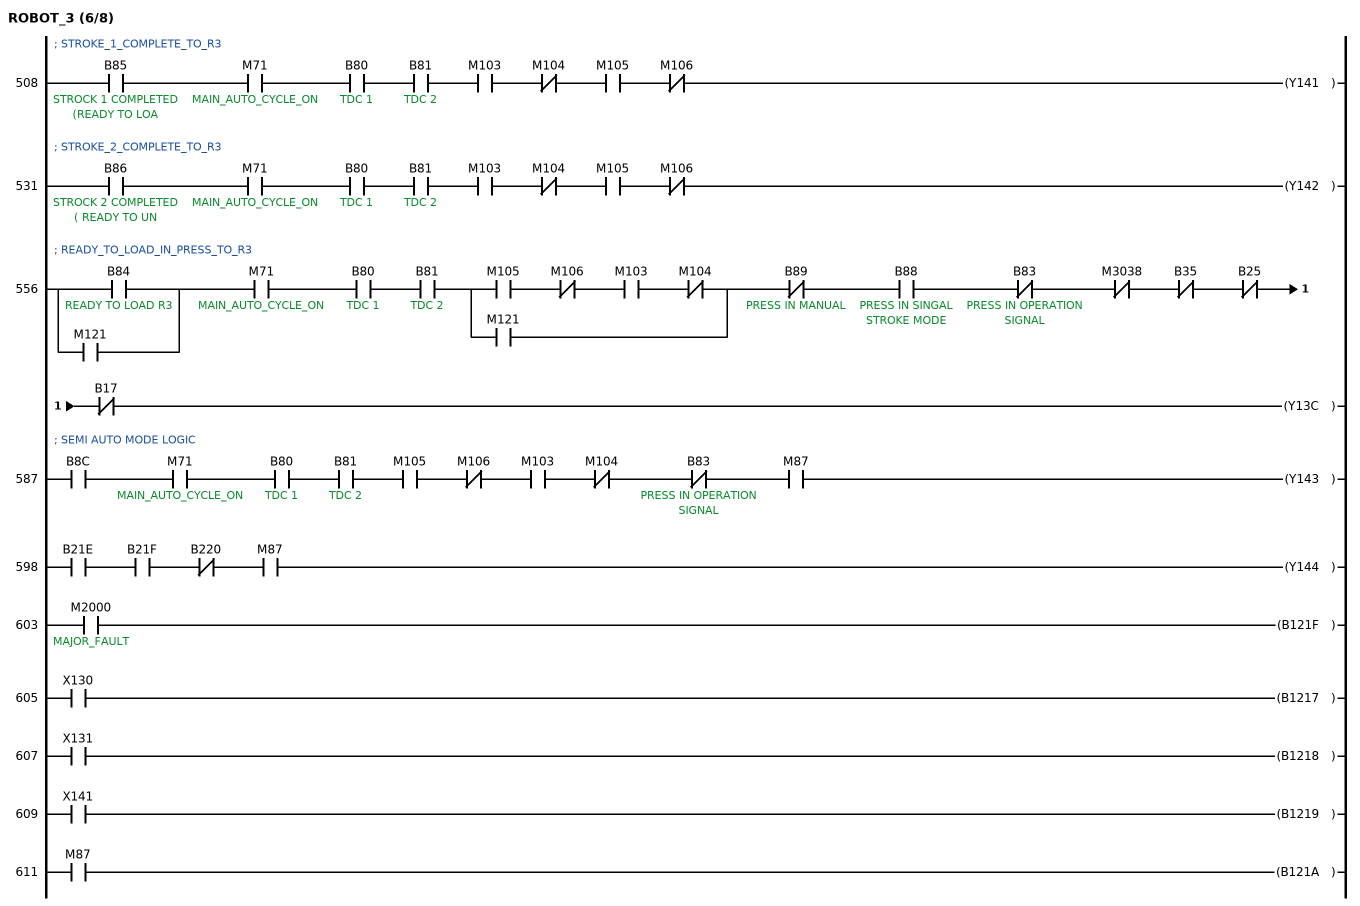
[picture p48: ladder of ROBOT_3, rungs at steps 508 to 611]
; STROKE_1_COMPLETE_TO_R3
508   LD      B85  ; STROCK 1 COMPLETED (READY TO LOA
      AND     M71  ; MAIN_AUTO_CYCLE_ON
      AND     B80  ; TDC 1
      AND     B81  ; TDC 2
      AND     M103
      ANI     M104
      AND     M105
      ANI     M106
      OUT     Y141
; STROKE_2_COMPLETE_TO_R3
531   LD      B86  ; STROCK 2 COMPLETED ( READY TO UN
      AND     M71  ; MAIN_AUTO_CYCLE_ON
      AND     B80  ; TDC 1
      AND     B81  ; TDC 2
      AND     M103
      ANI     M104
      AND     M105
      ANI     M106
      OUT     Y142
; READY_TO_LOAD_IN_PRESS_TO_R3
556   LD      B84  ; READY TO LOAD R3
      OR      M121
      AND     M71  ; MAIN_AUTO_CYCLE_ON
      AND     B80  ; TDC 1
      AND     B81  ; TDC 2
      LD      M105
      ANI     M106
      AND     M103
      ANI     M104
      OR      M121
      ANB
      ANI     B89  ; PRESS IN MANUAL
      AND     B88  ; PRESS IN SINGAL STROKE MODE
      ANI     B83  ; PRESS IN OPERATION SIGNAL
      ANI     M3038
      ANI     B35
      ANI     B25
      ANI     B17
      OUT     Y13C
; SEMI AUTO MODE LOGIC
587   LD      B8C
      AND     M71  ; MAIN_AUTO_CYCLE_ON
      AND     B80  ; TDC 1
      AND     B81  ; TDC 2
      AND     M105
      ANI     M106
      AND     M103
      ANI     M104
      ANI     B83  ; PRESS IN OPERATION SIGNAL
      AND     M87
      OUT     Y143
598   LD      B21E
      AND     B21F
      ANI     B220
      AND     M87
      OUT     Y144
603   LD      M2000  ; MAJOR_FAULT
      OUT     B121F
605   LD      X130
      OUT     B1217
607   LD      X131
      OUT     B1218
609   LD      X141
      OUT     B1219
611   LD      M87
      OUT     B121A
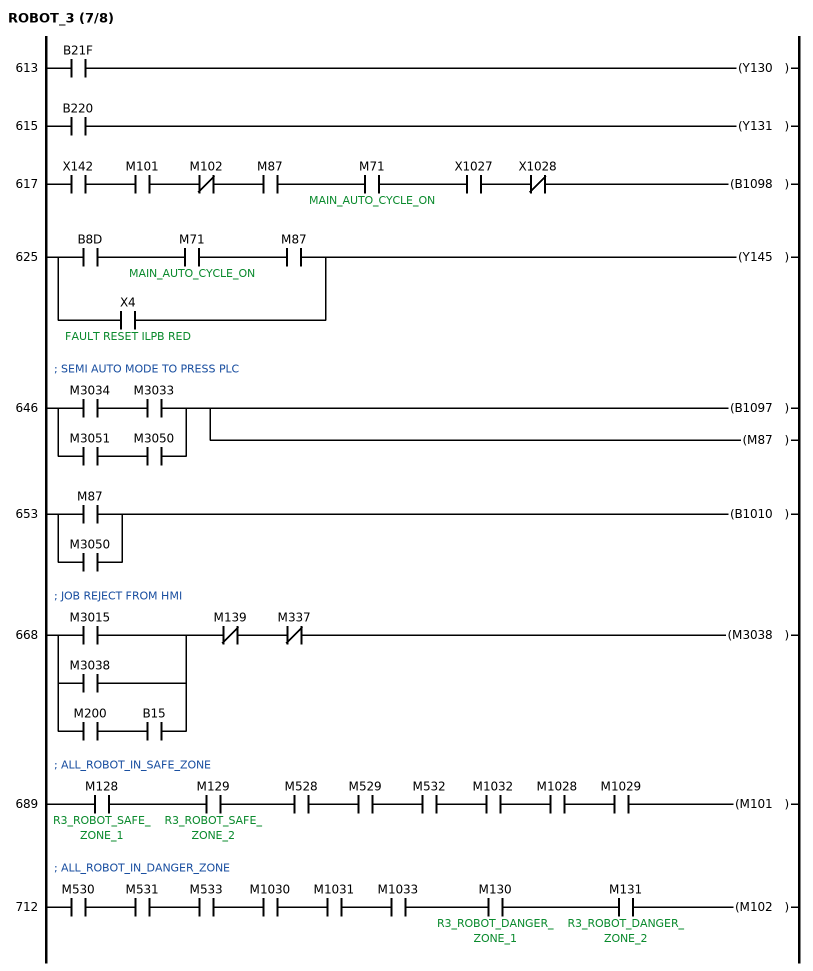
613   LD      B21F
      OUT     Y130
615   LD      B220
      OUT     Y131
617   LD      X142
      AND     M101
      ANI     M102
      AND     M87
      AND     M71  ; MAIN_AUTO_CYCLE_ON
      AND     X1027
      ANI     X1028
      OUT     B1098
625   LD      B8D
      AND     M71  ; MAIN_AUTO_CYCLE_ON
      AND     M87
      OR      X4  ; FAULT RESET ILPB RED
      OUT     Y145
; SEMI AUTO MODE TO PRESS PLC
646   LD      M3034
      AND     M3033
      LD      M3051
      AND     M3050
      ORB
      OUT     B1097
      OUT     M87
653   LD      M87
      OR      M3050
      OUT     B1010
; JOB REJECT FROM HMI
668   LD      M3015
      OR      M3038
      LD      M200
      AND     B15
      ORB
      ANI     M139
      ANI     M337
      OUT     M3038
; ALL_ROBOT_IN_SAFE_ZONE
689   LD      M128  ; R3_ROBOT_SAFE_ZONE_1
      AND     M129  ; R3_ROBOT_SAFE_ZONE_2
      AND     M528
      AND     M529
      AND     M532
      AND     M1032
      AND     M1028
      AND     M1029
      OUT     M101
; ALL_ROBOT_IN_DANGER_ZONE
712   LD      M530
      AND     M531
      AND     M533
      AND     M1030
      AND     M1031
      AND     M1033
      AND     M130  ; R3_ROBOT_DANGER_ZONE_1
      AND     M131  ; R3_ROBOT_DANGER_ZONE_2
      OUT     M102
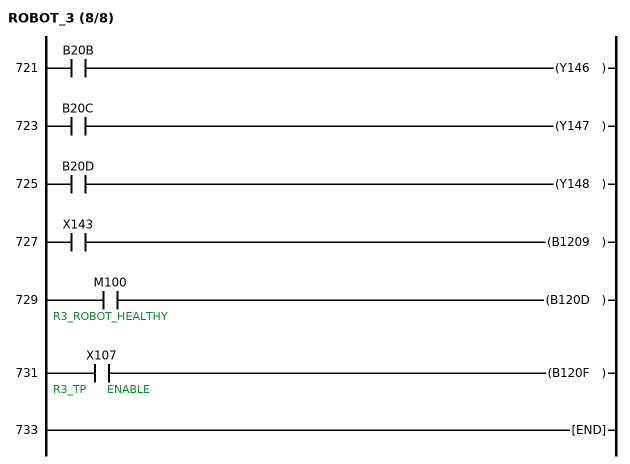
721   LD      B20B
      OUT     Y146
723   LD      B20C
      OUT     Y147
725   LD      B20D
      OUT     Y148
727   LD      X143
      OUT     B1209
729   LD      M100  ; R3_ROBOT_HEALTHY
      OUT     B120D
731   LD      X107  ; R3_TP      ENABLE
      OUT     B120F
733   END
END_PROGRAM

PROGRAM ROBOT_4
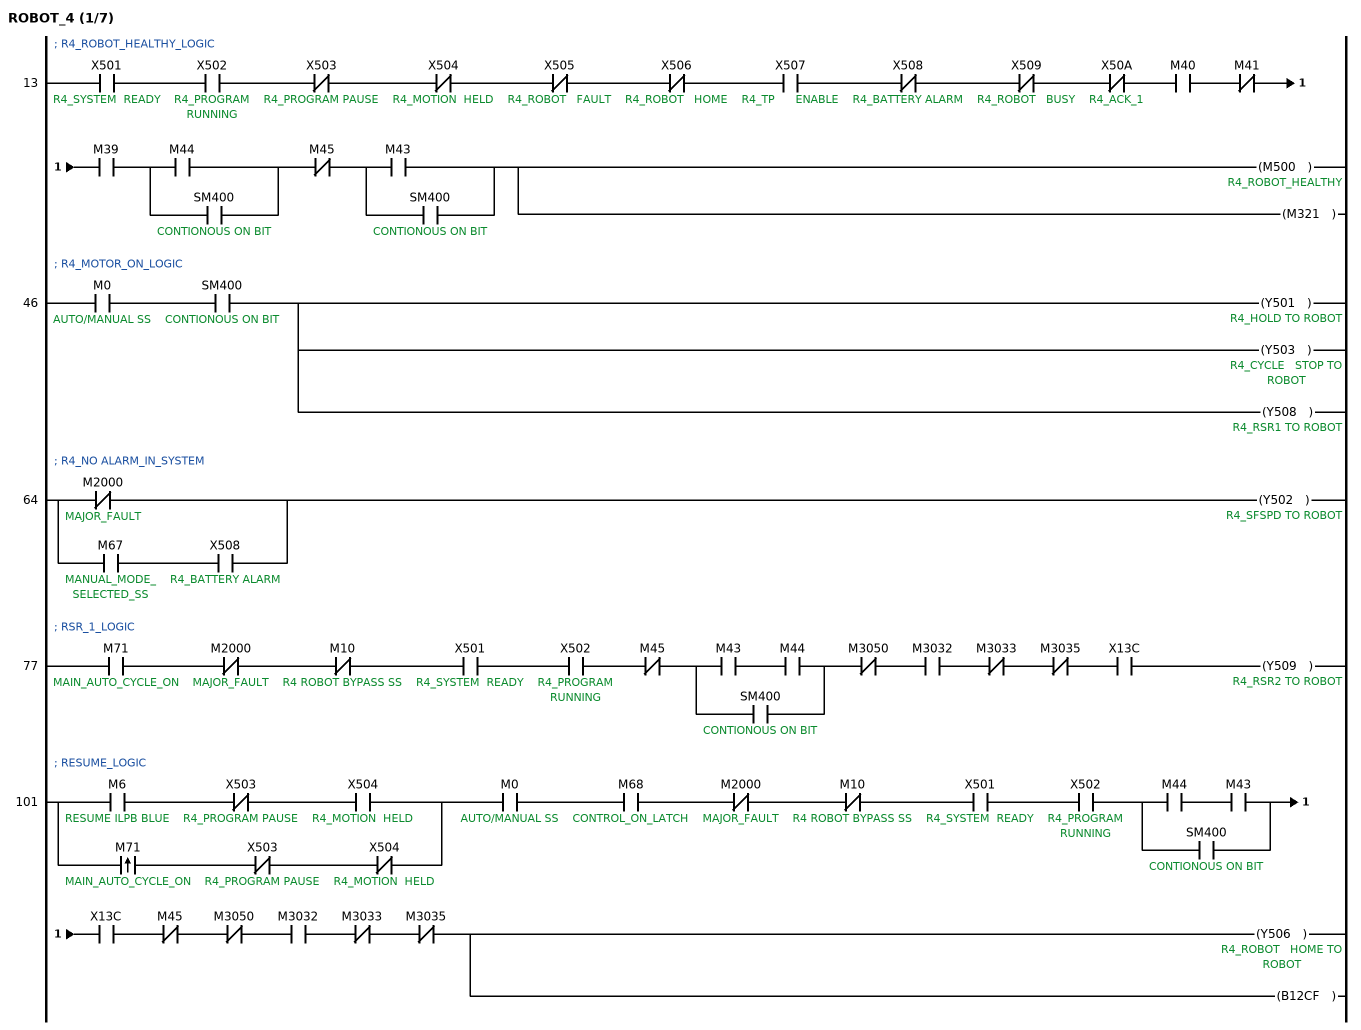
; R4_ROBOT_HEALTHY_LOGIC
13    LD      X501  ; R4_SYSTEM  READY
      AND     X502  ; R4_PROGRAM RUNNING
      ANI     X503  ; R4_PROGRAM PAUSE
      ANI     X504  ; R4_MOTION  HELD
      ANI     X505  ; R4_ROBOT   FAULT
      ANI     X506  ; R4_ROBOT   HOME
      AND     X507  ; R4_TP      ENABLE
      ANI     X508  ; R4_BATTERY ALARM
      ANI     X509  ; R4_ROBOT   BUSY
      ANI     X50A  ; R4_ACK_1
      AND     M40
      ANI     M41
      AND     M39
      LD      M44
      OR      SM400  ; CONTIONOUS ON BIT
      ANB
      ANI     M45
      LD      M43
      OR      SM400  ; CONTIONOUS ON BIT
      ANB
      OUT     M500  ; R4_ROBOT_HEALTHY
      OUT     M321
; R4_MOTOR_ON_LOGIC
46    LD      M0  ; AUTO/MANUAL SS
      AND     SM400  ; CONTIONOUS ON BIT
      OUT     Y501  ; R4_HOLD TO ROBOT
      OUT     Y503  ; R4_CYCLE   STOP TO ROBOT
      OUT     Y508  ; R4_RSR1 TO ROBOT
; R4_NO ALARM_IN_SYSTEM
64    LDI     M2000  ; MAJOR_FAULT
      LD      M67  ; MANUAL_MODE_SELECTED_SS
      AND     X508  ; R4_BATTERY ALARM
      ORB
      OUT     Y502  ; R4_SFSPD TO ROBOT
; RSR_1_LOGIC
77    LD      M71  ; MAIN_AUTO_CYCLE_ON
      ANI     M2000  ; MAJOR_FAULT
      ANI     M10  ; R4 ROBOT BYPASS SS
      AND     X501  ; R4_SYSTEM  READY
      AND     X502  ; R4_PROGRAM RUNNING
      ANI     M45
      LD      M43
      AND     M44
      OR      SM400  ; CONTIONOUS ON BIT
      ANB
      ANI     M3050
      AND     M3032
      ANI     M3033
      ANI     M3035
      AND     X13C
      OUT     Y509  ; R4_RSR2 TO ROBOT
; RESUME_LOGIC
101   LD      M6  ; RESUME ILPB BLUE
      ANI     X503  ; R4_PROGRAM PAUSE
      AND     X504  ; R4_MOTION  HELD
      LDP     M71  ; MAIN_AUTO_CYCLE_ON
      ANI     X503  ; R4_PROGRAM PAUSE
      ANI     X504  ; R4_MOTION  HELD
      ORB
      AND     M0  ; AUTO/MANUAL SS
      AND     M68  ; CONTROL_ON_LATCH
      ANI     M2000  ; MAJOR_FAULT
      ANI     M10  ; R4 ROBOT BYPASS SS
      AND     X501  ; R4_SYSTEM  READY
      AND     X502  ; R4_PROGRAM RUNNING
      LD      M44
      AND     M43
      OR      SM400  ; CONTIONOUS ON BIT
      ANB
      AND     X13C
      ANI     M45
      ANI     M3050
      AND     M3032
      ANI     M3033
      ANI     M3035
      OUT     Y506  ; R4_ROBOT   HOME TO ROBOT
      OUT     B12CF
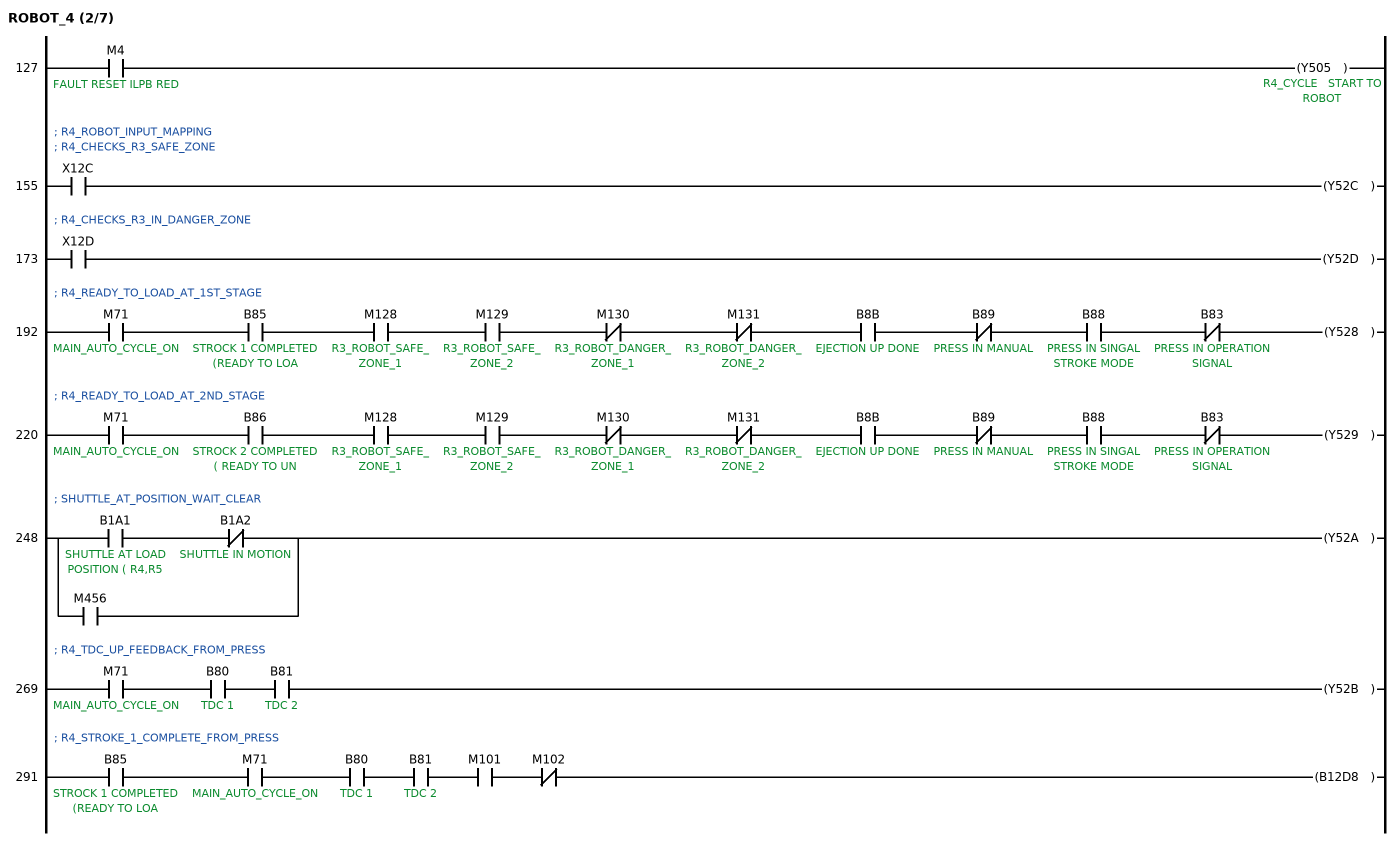
127   LD      M4  ; FAULT RESET ILPB RED
      OUT     Y505  ; R4_CYCLE   START TO ROBOT
; R4_ROBOT_INPUT_MAPPING
; R4_CHECKS_R3_SAFE_ZONE
155   LD      X12C
      OUT     Y52C
; R4_CHECKS_R3_IN_DANGER_ZONE
173   LD      X12D
      OUT     Y52D
; R4_READY_TO_LOAD_AT_1ST_STAGE
192   LD      M71  ; MAIN_AUTO_CYCLE_ON
      AND     B85  ; STROCK 1 COMPLETED (READY TO LOA
      AND     M128  ; R3_ROBOT_SAFE_ZONE_1
      AND     M129  ; R3_ROBOT_SAFE_ZONE_2
      ANI     M130  ; R3_ROBOT_DANGER_ZONE_1
      ANI     M131  ; R3_ROBOT_DANGER_ZONE_2
      AND     B8B  ; EJECTION UP DONE
      ANI     B89  ; PRESS IN MANUAL
      AND     B88  ; PRESS IN SINGAL STROKE MODE
      ANI     B83  ; PRESS IN OPERATION SIGNAL
      OUT     Y528
; R4_READY_TO_LOAD_AT_2ND_STAGE
220   LD      M71  ; MAIN_AUTO_CYCLE_ON
      AND     B86  ; STROCK 2 COMPLETED ( READY TO UN
      AND     M128  ; R3_ROBOT_SAFE_ZONE_1
      AND     M129  ; R3_ROBOT_SAFE_ZONE_2
      ANI     M130  ; R3_ROBOT_DANGER_ZONE_1
      ANI     M131  ; R3_ROBOT_DANGER_ZONE_2
      AND     B8B  ; EJECTION UP DONE
      ANI     B89  ; PRESS IN MANUAL
      AND     B88  ; PRESS IN SINGAL STROKE MODE
      ANI     B83  ; PRESS IN OPERATION SIGNAL
      OUT     Y529
; SHUTTLE_AT_POSITION_WAIT_CLEAR
248   LD      B1A1  ; SHUTTLE AT LOAD POSITION ( R4,R5
      ANI     B1A2  ; SHUTTLE IN MOTION
      OR      M456
      OUT     Y52A
; R4_TDC_UP_FEEDBACK_FROM_PRESS
269   LD      M71  ; MAIN_AUTO_CYCLE_ON
      AND     B80  ; TDC 1
      AND     B81  ; TDC 2
      OUT     Y52B
; R4_STROKE_1_COMPLETE_FROM_PRESS
291   LD      B85  ; STROCK 1 COMPLETED (READY TO LOA
      AND     M71  ; MAIN_AUTO_CYCLE_ON
      AND     B80  ; TDC 1
      AND     B81  ; TDC 2
      AND     M101
      ANI     M102
      OUT     B12D8
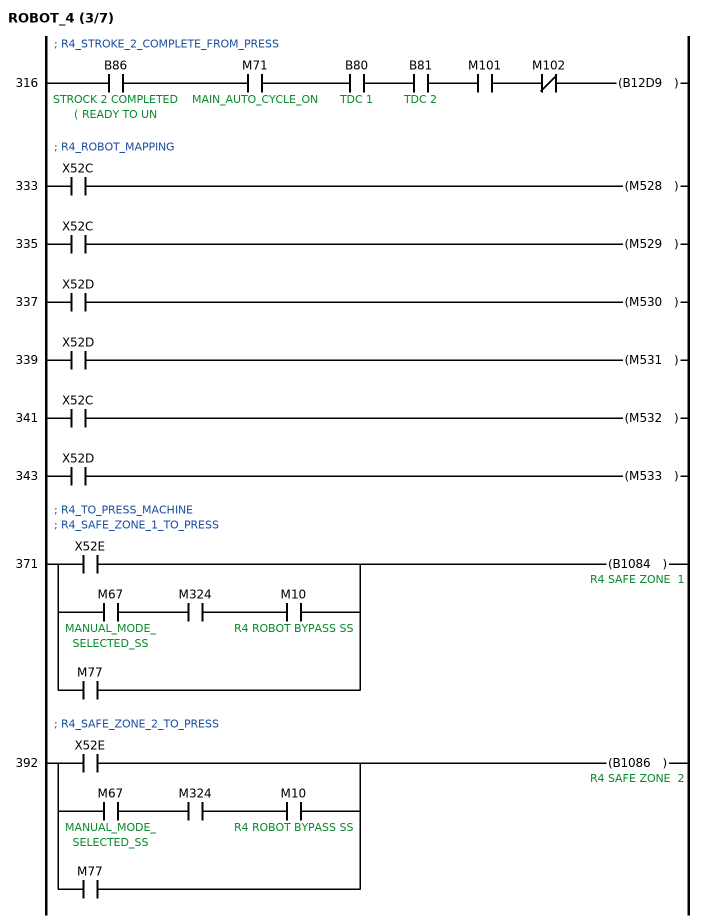
; R4_STROKE_2_COMPLETE_FROM_PRESS
316   LD      B86  ; STROCK 2 COMPLETED ( READY TO UN
      AND     M71  ; MAIN_AUTO_CYCLE_ON
      AND     B80  ; TDC 1
      AND     B81  ; TDC 2
      AND     M101
      ANI     M102
      OUT     B12D9
; R4_ROBOT_MAPPING
333   LD      X52C
      OUT     M528
335   LD      X52C
      OUT     M529
337   LD      X52D
      OUT     M530
339   LD      X52D
      OUT     M531
341   LD      X52C
      OUT     M532
343   LD      X52D
      OUT     M533
; R4_TO_PRESS_MACHINE
; R4_SAFE_ZONE_1_TO_PRESS
371   LD      X52E
      LD      M67  ; MANUAL_MODE_SELECTED_SS
      AND     M324
      AND     M10  ; R4 ROBOT BYPASS SS
      ORB
      OR      M77
      OUT     B1084  ; R4 SAFE ZONE  1
; R4_SAFE_ZONE_2_TO_PRESS
392   LD      X52E
      LD      M67  ; MANUAL_MODE_SELECTED_SS
      AND     M324
      AND     M10  ; R4 ROBOT BYPASS SS
      ORB
      OR      M77
      OUT     B1086  ; R4 SAFE ZONE  2
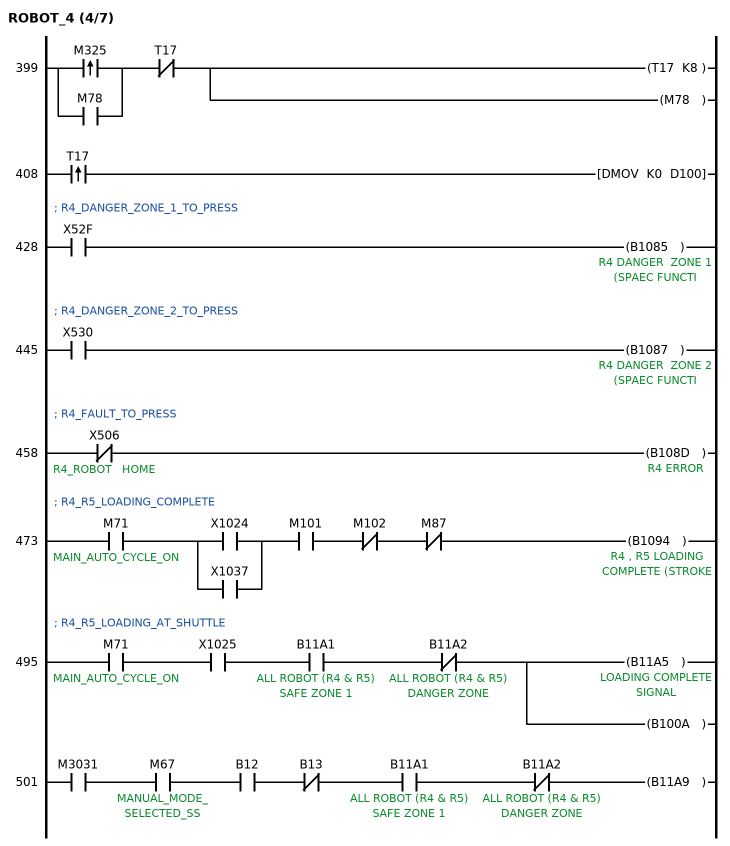
399   LDP     M325
      OR      M78
      ANI     T17
      OUT     T17 K8
      OUT     M78
408   LDP     T17
      DMOV    K0 D100
; R4_DANGER_ZONE_1_TO_PRESS
428   LD      X52F
      OUT     B1085  ; R4 DANGER  ZONE 1 (SPAEC FUNCTI
; R4_DANGER_ZONE_2_TO_PRESS
445   LD      X530
      OUT     B1087  ; R4 DANGER  ZONE 2 (SPAEC FUNCTI
; R4_FAULT_TO_PRESS
458   LDI     X506  ; R4_ROBOT   HOME
      OUT     B108D  ; R4 ERROR
; R4_R5_LOADING_COMPLETE
473   LD      M71  ; MAIN_AUTO_CYCLE_ON
      LD      X1024
      OR      X1037
      ANB
      AND     M101
      ANI     M102
      ANI     M87
      OUT     B1094  ; R4 , R5 LOADING COMPLETE (STROKE
; R4_R5_LOADING_AT_SHUTTLE
495   LD      M71  ; MAIN_AUTO_CYCLE_ON
      AND     X1025
      AND     B11A1  ; ALL ROBOT (R4 & R5) SAFE ZONE 1
      ANI     B11A2  ; ALL ROBOT (R4 & R5) DANGER ZONE
      OUT     B11A5  ; LOADING COMPLETE SIGNAL
      OUT     B100A
501   LD      M3031
      AND     M67  ; MANUAL_MODE_SELECTED_SS
      AND     B12
      ANI     B13
      AND     B11A1  ; ALL ROBOT (R4 & R5) SAFE ZONE 1
      ANI     B11A2  ; ALL ROBOT (R4 & R5) DANGER ZONE
      OUT     B11A9
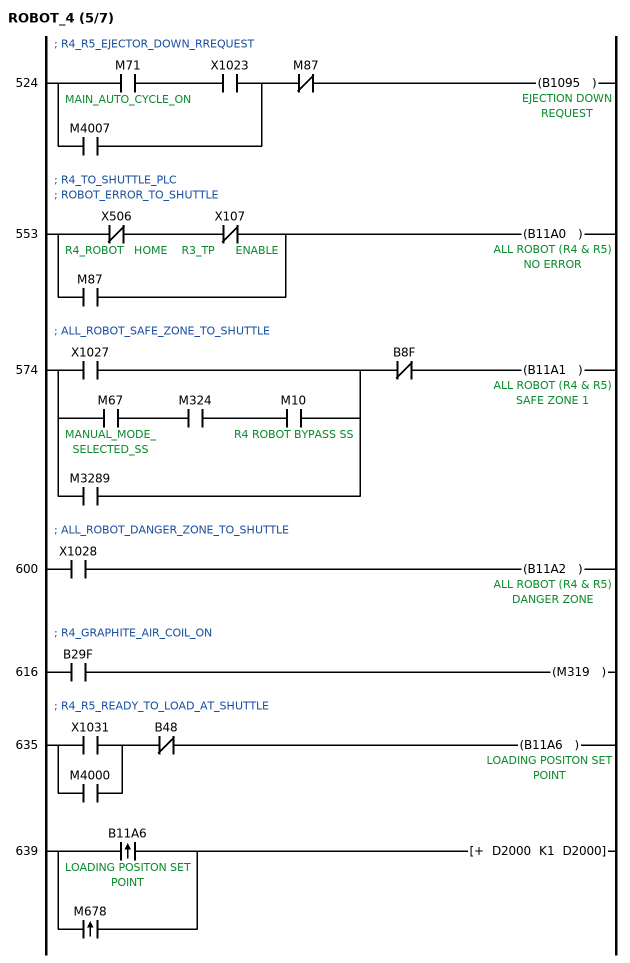
; R4_R5_EJECTOR_DOWN_RREQUEST
524   LD      M71  ; MAIN_AUTO_CYCLE_ON
      AND     X1023
      OR      M4007
      ANI     M87
      OUT     B1095  ; EJECTION DOWN REQUEST
; R4_TO_SHUTTLE_PLC
; ROBOT_ERROR_TO_SHUTTLE
553   LDI     X506  ; R4_ROBOT   HOME
      ANI     X107  ; R3_TP      ENABLE
      OR      M87
      OUT     B11A0  ; ALL ROBOT (R4 & R5) NO ERROR
; ALL_ROBOT_SAFE_ZONE_TO_SHUTTLE
574   LD      X1027
      LD      M67  ; MANUAL_MODE_SELECTED_SS
      AND     M324
      AND     M10  ; R4 ROBOT BYPASS SS
      ORB
      OR      M3289
      ANI     B8F
      OUT     B11A1  ; ALL ROBOT (R4 & R5) SAFE ZONE 1
; ALL_ROBOT_DANGER_ZONE_TO_SHUTTLE
600   LD      X1028
      OUT     B11A2  ; ALL ROBOT (R4 & R5) DANGER ZONE
; R4_GRAPHITE_AIR_COIL_ON
616   LD      B29F
      OUT     M319
; R4_R5_READY_TO_LOAD_AT_SHUTTLE
635   LD      X1031
      OR      M4000
      ANI     B48
      OUT     B11A6  ; LOADING POSITON SET POINT
639   LDP     B11A6  ; LOADING POSITON SET POINT
      ORP     M678
      +       D2000 K1 D2000
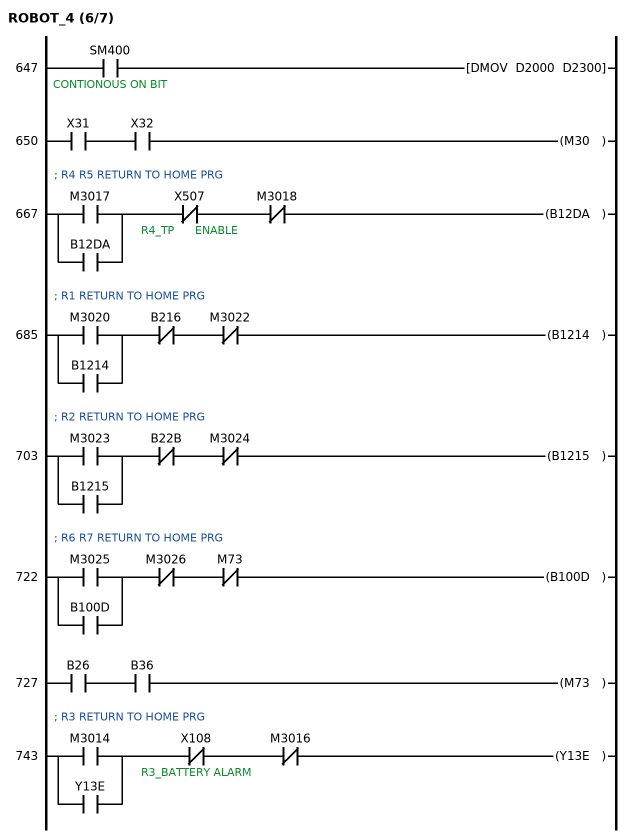
647   LD      SM400  ; CONTIONOUS ON BIT
      DMOV    D2000 D2300
650   LD      X31
      AND     X32
      OUT     M30
; R4 R5 RETURN TO HOME PRG
667   LD      M3017
      OR      B12DA
      ANI     X507  ; R4_TP      ENABLE
      ANI     M3018
      OUT     B12DA
; R1 RETURN TO HOME PRG
685   LD      M3020
      OR      B1214
      ANI     B216
      ANI     M3022
      OUT     B1214
; R2 RETURN TO HOME PRG
703   LD      M3023
      OR      B1215
      ANI     B22B
      ANI     M3024
      OUT     B1215
; R6 R7 RETURN TO HOME PRG
722   LD      M3025
      OR      B100D
      ANI     M3026
      ANI     M73
      OUT     B100D
727   LD      B26
      AND     B36
      OUT     M73
; R3 RETURN TO HOME PRG
743   LD      M3014
      OR      Y13E
      ANI     X108  ; R3_BATTERY ALARM
      ANI     M3016
      OUT     Y13E
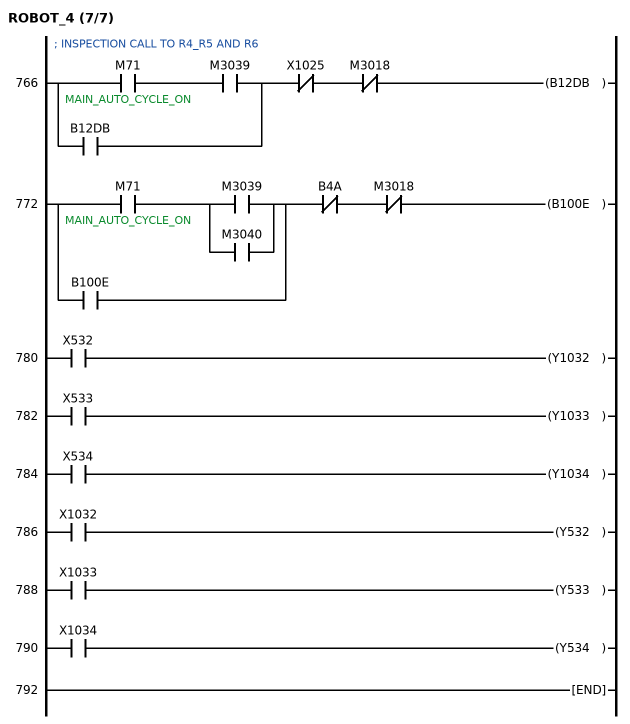
; INSPECTION CALL TO R4_R5 AND R6
766   LD      M71  ; MAIN_AUTO_CYCLE_ON
      AND     M3039
      OR      B12DB
      ANI     X1025
      ANI     M3018
      OUT     B12DB
772   LD      M71  ; MAIN_AUTO_CYCLE_ON
      LD      M3039
      OR      M3040
      ANB
      OR      B100E
      ANI     B4A
      ANI     M3018
      OUT     B100E
780   LD      X532
      OUT     Y1032
782   LD      X533
      OUT     Y1033
784   LD      X534
      OUT     Y1034
786   LD      X1032
      OUT     Y532
788   LD      X1033
      OUT     Y533
790   LD      X1034
      OUT     Y534
792   END
END_PROGRAM

PROGRAM ROBOT_5
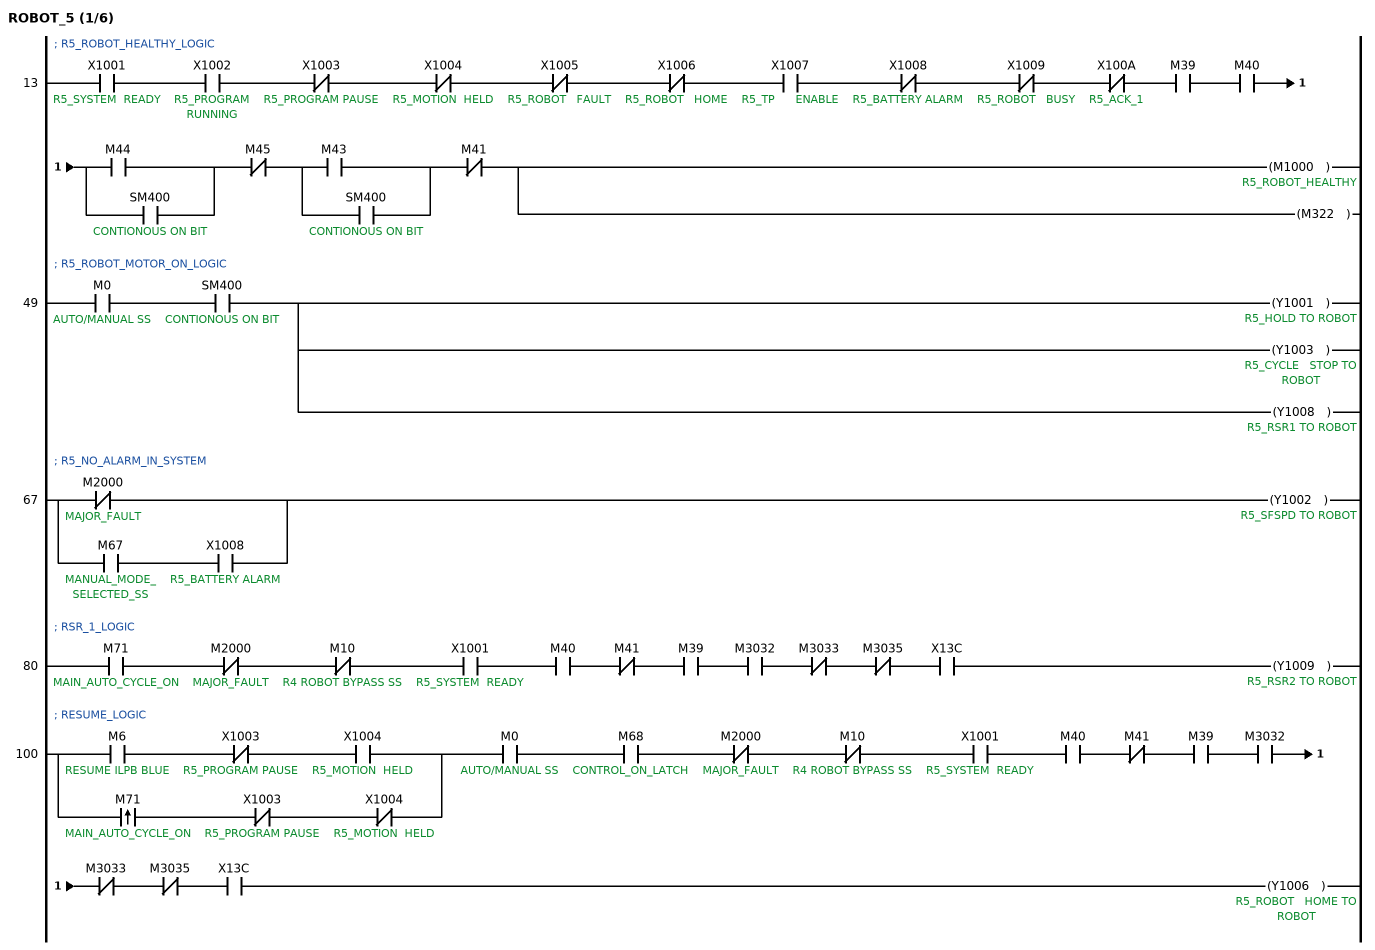
; R5_ROBOT_HEALTHY_LOGIC
13    LD      X1001  ; R5_SYSTEM  READY
      AND     X1002  ; R5_PROGRAM RUNNING
      ANI     X1003  ; R5_PROGRAM PAUSE
      ANI     X1004  ; R5_MOTION  HELD
      ANI     X1005  ; R5_ROBOT   FAULT
      ANI     X1006  ; R5_ROBOT   HOME
      AND     X1007  ; R5_TP      ENABLE
      ANI     X1008  ; R5_BATTERY ALARM
      ANI     X1009  ; R5_ROBOT   BUSY
      ANI     X100A  ; R5_ACK_1
      AND     M39
      AND     M40
      LD      M44
      OR      SM400  ; CONTIONOUS ON BIT
      ANB
      ANI     M45
      LD      M43
      OR      SM400  ; CONTIONOUS ON BIT
      ANB
      ANI     M41
      OUT     M1000  ; R5_ROBOT_HEALTHY
      OUT     M322
; R5_ROBOT_MOTOR_ON_LOGIC
49    LD      M0  ; AUTO/MANUAL SS
      AND     SM400  ; CONTIONOUS ON BIT
      OUT     Y1001  ; R5_HOLD TO ROBOT
      OUT     Y1003  ; R5_CYCLE   STOP TO ROBOT
      OUT     Y1008  ; R5_RSR1 TO ROBOT
; R5_NO_ALARM_IN_SYSTEM
67    LDI     M2000  ; MAJOR_FAULT
      LD      M67  ; MANUAL_MODE_SELECTED_SS
      AND     X1008  ; R5_BATTERY ALARM
      ORB
      OUT     Y1002  ; R5_SFSPD TO ROBOT
; RSR_1_LOGIC
80    LD      M71  ; MAIN_AUTO_CYCLE_ON
      ANI     M2000  ; MAJOR_FAULT
      ANI     M10  ; R4 ROBOT BYPASS SS
      AND     X1001  ; R5_SYSTEM  READY
      AND     M40
      ANI     M41
      AND     M39
      AND     M3032
      ANI     M3033
      ANI     M3035
      AND     X13C
      OUT     Y1009  ; R5_RSR2 TO ROBOT
; RESUME_LOGIC
100   LD      M6  ; RESUME ILPB BLUE
      ANI     X1003  ; R5_PROGRAM PAUSE
      AND     X1004  ; R5_MOTION  HELD
      LDP     M71  ; MAIN_AUTO_CYCLE_ON
      ANI     X1003  ; R5_PROGRAM PAUSE
      ANI     X1004  ; R5_MOTION  HELD
      ORB
      AND     M0  ; AUTO/MANUAL SS
      AND     M68  ; CONTROL_ON_LATCH
      ANI     M2000  ; MAJOR_FAULT
      ANI     M10  ; R4 ROBOT BYPASS SS
      AND     X1001  ; R5_SYSTEM  READY
      AND     M40
      ANI     M41
      AND     M39
      AND     M3032
      ANI     M3033
      ANI     M3035
      AND     X13C
      OUT     Y1006  ; R5_ROBOT   HOME TO ROBOT
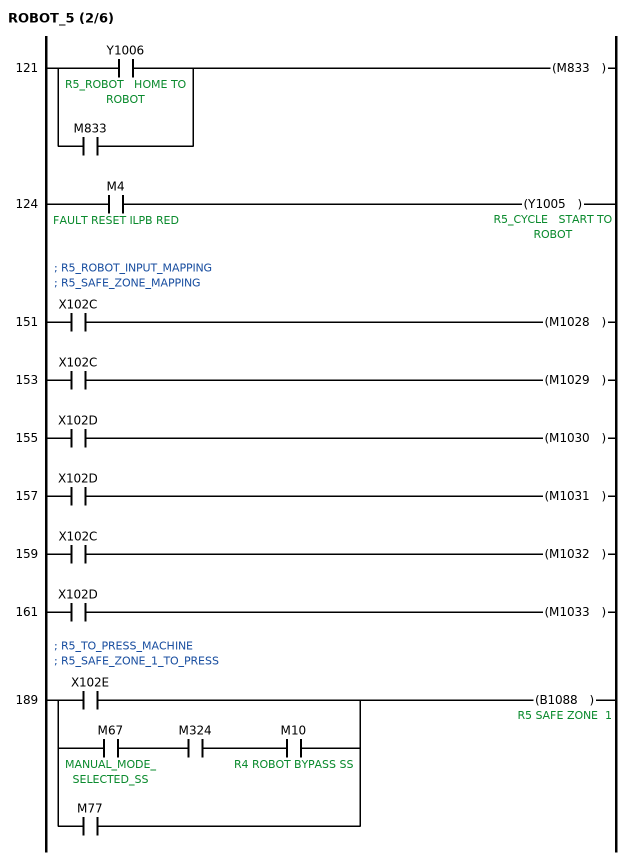
121   LD      Y1006  ; R5_ROBOT   HOME TO ROBOT
      OR      M833
      OUT     M833
124   LD      M4  ; FAULT RESET ILPB RED
      OUT     Y1005  ; R5_CYCLE   START TO ROBOT
; R5_ROBOT_INPUT_MAPPING
; R5_SAFE_ZONE_MAPPING
151   LD      X102C
      OUT     M1028
153   LD      X102C
      OUT     M1029
155   LD      X102D
      OUT     M1030
157   LD      X102D
      OUT     M1031
159   LD      X102C
      OUT     M1032
161   LD      X102D
      OUT     M1033
; R5_TO_PRESS_MACHINE
; R5_SAFE_ZONE_1_TO_PRESS
189   LD      X102E
      LD      M67  ; MANUAL_MODE_SELECTED_SS
      AND     M324
      AND     M10  ; R4 ROBOT BYPASS SS
      ORB
      OR      M77
      OUT     B1088  ; R5 SAFE ZONE  1
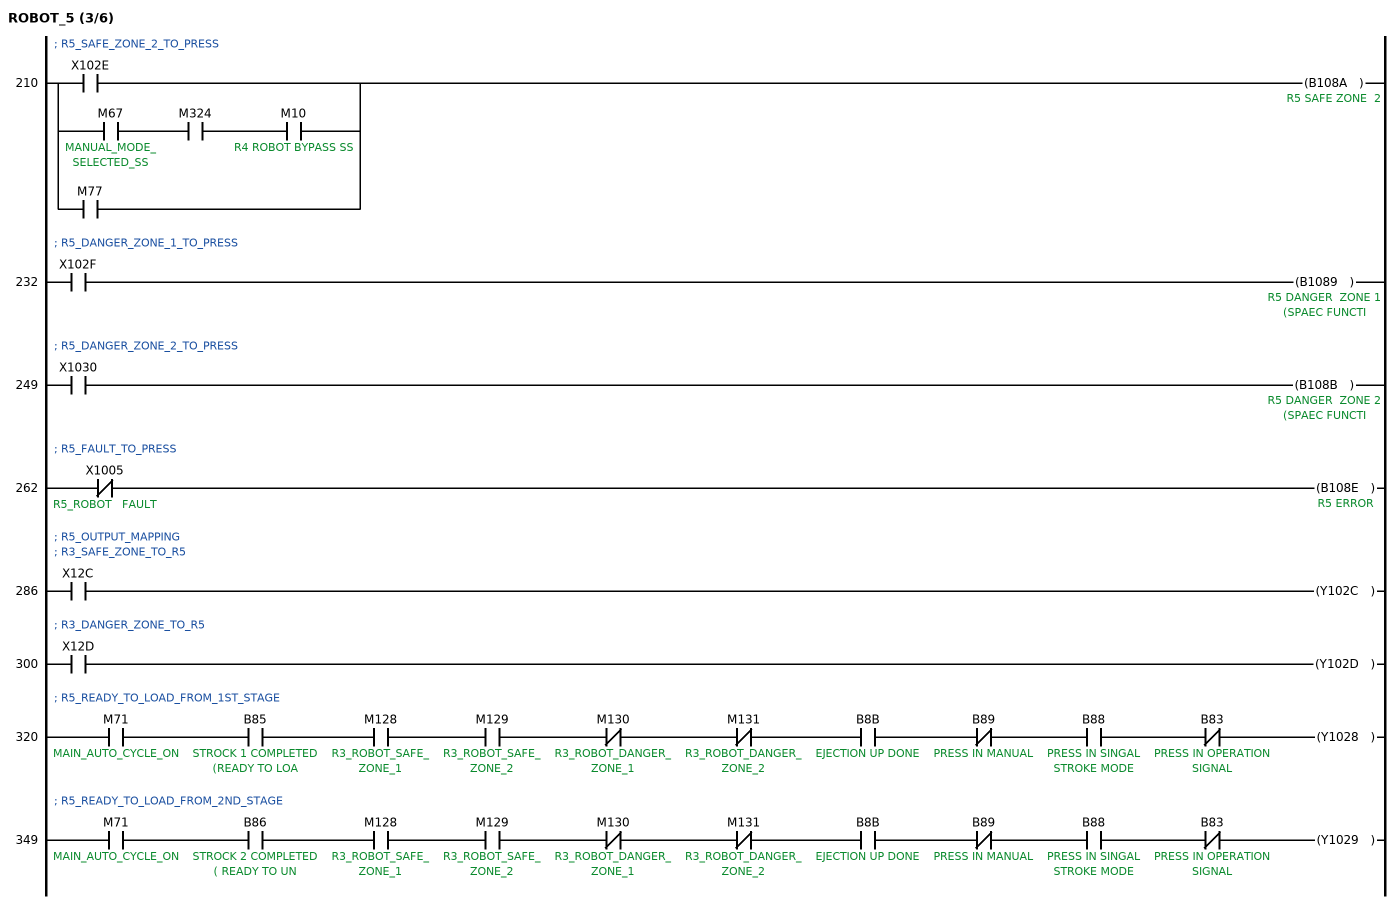
; R5_SAFE_ZONE_2_TO_PRESS
210   LD      X102E
      LD      M67  ; MANUAL_MODE_SELECTED_SS
      AND     M324
      AND     M10  ; R4 ROBOT BYPASS SS
      ORB
      OR      M77
      OUT     B108A  ; R5 SAFE ZONE  2
; R5_DANGER_ZONE_1_TO_PRESS
232   LD      X102F
      OUT     B1089  ; R5 DANGER  ZONE 1 (SPAEC FUNCTI
; R5_DANGER_ZONE_2_TO_PRESS
249   LD      X1030
      OUT     B108B  ; R5 DANGER  ZONE 2 (SPAEC FUNCTI
; R5_FAULT_TO_PRESS
262   LDI     X1005  ; R5_ROBOT   FAULT
      OUT     B108E  ; R5 ERROR
; R5_OUTPUT_MAPPING
; R3_SAFE_ZONE_TO_R5
286   LD      X12C
      OUT     Y102C
; R3_DANGER_ZONE_TO_R5
300   LD      X12D
      OUT     Y102D
; R5_READY_TO_LOAD_FROM_1ST_STAGE
320   LD      M71  ; MAIN_AUTO_CYCLE_ON
      AND     B85  ; STROCK 1 COMPLETED (READY TO LOA
      AND     M128  ; R3_ROBOT_SAFE_ZONE_1
      AND     M129  ; R3_ROBOT_SAFE_ZONE_2
      ANI     M130  ; R3_ROBOT_DANGER_ZONE_1
      ANI     M131  ; R3_ROBOT_DANGER_ZONE_2
      AND     B8B  ; EJECTION UP DONE
      ANI     B89  ; PRESS IN MANUAL
      AND     B88  ; PRESS IN SINGAL STROKE MODE
      ANI     B83  ; PRESS IN OPERATION SIGNAL
      OUT     Y1028
; R5_READY_TO_LOAD_FROM_2ND_STAGE
349   LD      M71  ; MAIN_AUTO_CYCLE_ON
      AND     B86  ; STROCK 2 COMPLETED ( READY TO UN
      AND     M128  ; R3_ROBOT_SAFE_ZONE_1
      AND     M129  ; R3_ROBOT_SAFE_ZONE_2
      ANI     M130  ; R3_ROBOT_DANGER_ZONE_1
      ANI     M131  ; R3_ROBOT_DANGER_ZONE_2
      AND     B8B  ; EJECTION UP DONE
      ANI     B89  ; PRESS IN MANUAL
      AND     B88  ; PRESS IN SINGAL STROKE MODE
      ANI     B83  ; PRESS IN OPERATION SIGNAL
      OUT     Y1029
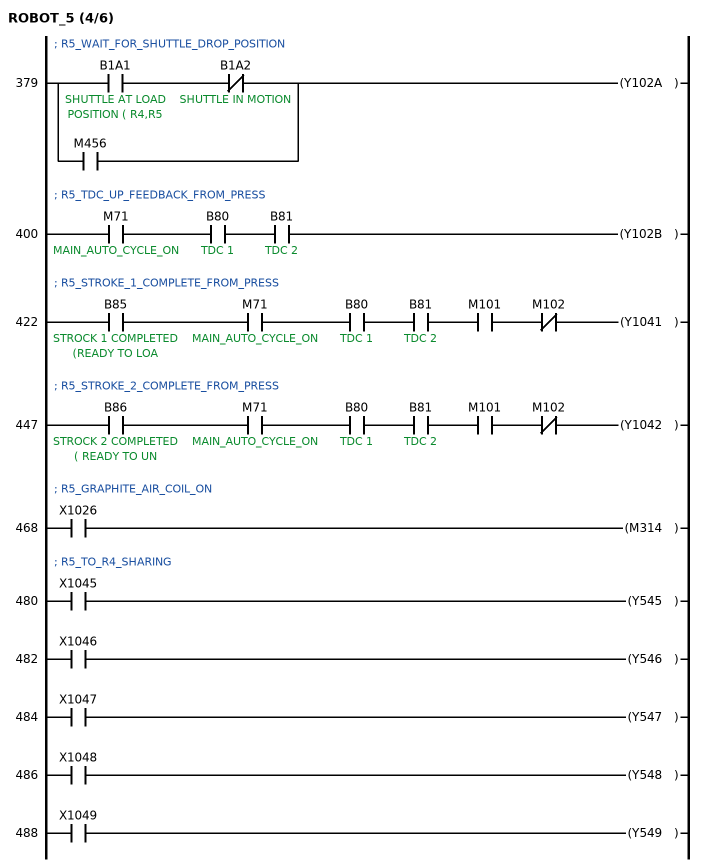
; R5_WAIT_FOR_SHUTTLE_DROP_POSITION
379   LD      B1A1  ; SHUTTLE AT LOAD POSITION ( R4,R5
      ANI     B1A2  ; SHUTTLE IN MOTION
      OR      M456
      OUT     Y102A
; R5_TDC_UP_FEEDBACK_FROM_PRESS
400   LD      M71  ; MAIN_AUTO_CYCLE_ON
      AND     B80  ; TDC 1
      AND     B81  ; TDC 2
      OUT     Y102B
; R5_STROKE_1_COMPLETE_FROM_PRESS
422   LD      B85  ; STROCK 1 COMPLETED (READY TO LOA
      AND     M71  ; MAIN_AUTO_CYCLE_ON
      AND     B80  ; TDC 1
      AND     B81  ; TDC 2
      AND     M101
      ANI     M102
      OUT     Y1041
; R5_STROKE_2_COMPLETE_FROM_PRESS
447   LD      B86  ; STROCK 2 COMPLETED ( READY TO UN
      AND     M71  ; MAIN_AUTO_CYCLE_ON
      AND     B80  ; TDC 1
      AND     B81  ; TDC 2
      AND     M101
      ANI     M102
      OUT     Y1042
; R5_GRAPHITE_AIR_COIL_ON
468   LD      X1026
      OUT     M314
; R5_TO_R4_SHARING
480   LD      X1045
      OUT     Y545
482   LD      X1046
      OUT     Y546
484   LD      X1047
      OUT     Y547
486   LD      X1048
      OUT     Y548
488   LD      X1049
      OUT     Y549
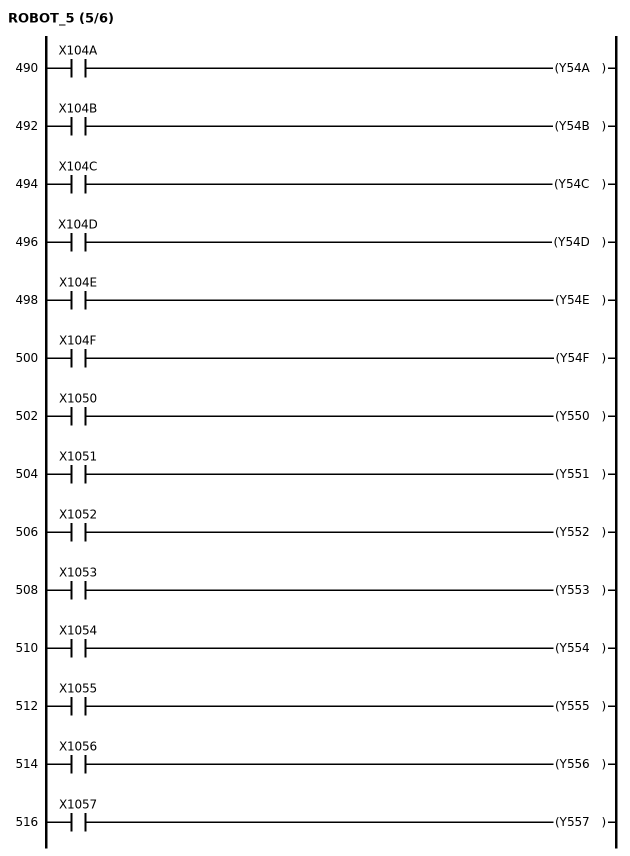
490   LD      X104A
      OUT     Y54A
492   LD      X104B
      OUT     Y54B
494   LD      X104C
      OUT     Y54C
496   LD      X104D
      OUT     Y54D
498   LD      X104E
      OUT     Y54E
500   LD      X104F
      OUT     Y54F
502   LD      X1050
      OUT     Y550
504   LD      X1051
      OUT     Y551
506   LD      X1052
      OUT     Y552
508   LD      X1053
      OUT     Y553
510   LD      X1054
      OUT     Y554
512   LD      X1055
      OUT     Y555
514   LD      X1056
      OUT     Y556
516   LD      X1057
      OUT     Y557
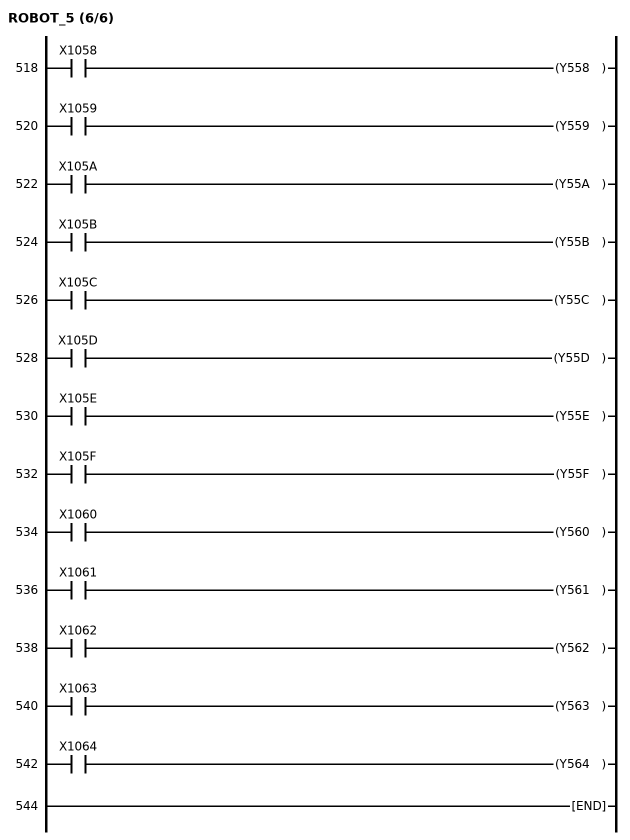
518   LD      X1058
      OUT     Y558
520   LD      X1059
      OUT     Y559
522   LD      X105A
      OUT     Y55A
524   LD      X105B
      OUT     Y55B
526   LD      X105C
      OUT     Y55C
528   LD      X105D
      OUT     Y55D
530   LD      X105E
      OUT     Y55E
532   LD      X105F
      OUT     Y55F
534   LD      X1060
      OUT     Y560
536   LD      X1061
      OUT     Y561
538   LD      X1062
      OUT     Y562
540   LD      X1063
      OUT     Y563
542   LD      X1064
      OUT     Y564
544   END
END_PROGRAM

// device comments not shown above
X100  ; R3_CMD     ENABLE
X101  ; R3_SYSTEM  READY
X10C  ; R3_ACK_3
X10D  ; R3_ACK_4
X10E  ; R3_ACK_5
X10F  ; R3_ACK_6
X110  ; R3_ACK_7
X111  ; R3_ACK_8
X112  ; R3_SNACK
X500  ; R4_CMD     ENABLE
X50B  ; R4_ACK_2
X50C  ; R4_ACK_3
X50D  ; R4_ACK_4
X50E  ; R4_ACK_5
X50F  ; R4_ACK_6
X510  ; R4_ACK_7
X511  ; R4_ACK_8
X512  ; R4_SNACK
X1000  ; R5_CMD     ENABLE
X100B  ; R5_ACK_2
X100C  ; R5_ACK_3
X100D  ; R5_ACK_4
X100E  ; R5_ACK_5
X100F  ; R5_ACK_6
X1010  ; R5_ACK_7
X1011  ; R5_ACK_8
X1012  ; R5_SNACK
Y100  ; R3_IMSTP   STOP
Y107  ; R3_ENABLE  TO ROBOT
Y10B  ; R3_RSR4 TO ROBOT
Y10D  ; R3_RSR6 TO ROBOT
Y10E  ; R3_RSR7 TO ROBOT
Y10F  ; R3_RSR8 TO ROBOT
Y110  ; R3_PNS     STROBE
Y111  ; R3_PRODUCTION START
Y500  ; R4_IMSTP   STOP
Y504  ; R4_FAULT   RESET TO ROBOT
Y507  ; R4_ENABLE  TO ROBOT
Y50A  ; R4_RSR3 TO ROBOT
Y50B  ; R4_RSR4 TO ROBOT
Y50C  ; R4_RSR5 TO ROBOT
Y50D  ; R4_RSR6 TO ROBOT
Y50E  ; R4_RSR7 TO ROBOT
Y50F  ; R4_RSR8 TO ROBOT
Y510  ; R4_PNS     STROBE
Y511  ; R4_PRODUCTION START
Y1000  ; R5_IMSTP   STOP
Y1004  ; R5_FAULT   RESET TO ROBOT
Y1007  ; R5_ENABLE  TO ROBOT
Y100A  ; R5_RSR3 TO ROBOT
Y100B  ; R5_RSR4 TO ROBOT
Y100C  ; R5_RSR5 TO ROBOT
Y100D  ; R5_RSR6 TO ROBOT
Y100E  ; R5_RSR7 TO ROBOT
Y100F  ; R5_RSR8 TO ROBOT
Y1010  ; R5_PNS     STROBE
Y1011  ; R5_PRODUCTION START
B8A  ; ROBOT REJECT
B1090  ; CYCLE SEMI-AUTO MODE
B1096  ; REJECT SELECTOR FEEDBACK
B11A7  ; UNLOADING POSITION SET POINT
